// TIA Portal V20 export
DATA_BLOCK "Global DB"   // DB7
{ S7_Optimized_Access := 'TRUE' }
// stored: MemoryReserve 100
   VAR
      Valve1 : "Equipment";
      Valve2 { S7_SetPoint := 'True'} : "Equipment";
      Valve3 { S7_SetPoint := 'True'} : "Equipment";
      Heater { S7_SetPoint := 'True'} : "Equipment";
      Mixer { S7_SetPoint := 'True'} : "Equipment";
      Process_Start { S7_SetPoint := 'True'} : Bool;
      Process_Stop : Bool;
      Process_Reset : Bool;
      Process_Step : Int;
      Process_Count : Int;
      isTankHeated : Bool;
      isTankMixed : Bool;
      Tank1 : "Tank";
      Tank2 { S7_SetPoint := 'True'} : "Tank";
      positive_edge { S7_SetPoint := 'True'} : Bool;
      prevLevel : DInt;
   END_VAR
BEGIN
   Heater."type" := 1;
   Mixer."type" := 2;
END_DATA_BLOCK
